// TIA Portal project "FactoryIO-ProductAllocate" (V17)

(* hardware
DEVICE "S71500/ET200MP-Station_1"  S7-1500 station
   slot 0: "Profilschiene_0"  6ES7 590-1***0-0AA0
   slot 1: "PLC_1"  CPU 1511-1 PN  6ES7 511-1AK00-0AB0  V1.8
   slot 2: "AI 8xU/I/RTD/TC ST_1"  AI 8xU/I/RTD/TC ST  6ES7 531-7KF00-0AB0  V2.0
   slot 3: "AI 8xU/I/RTD/TC ST_2"  AI 8xU/I/RTD/TC ST  6ES7 531-7KF00-0AB0  V2.0
   slot 4: "AI 8xU/I/RTD/TC ST_3"  AI 8xU/I/RTD/TC ST  6ES7 531-7KF00-0AB0  V2.0
   slot 5: "AI 8xU/I/RTD/TC ST_4"  AI 8xU/I/RTD/TC ST  6ES7 531-7KF00-0AB0  V2.0
   slot 6: "DI 16x24VDC BA_1"  DI 16x24VDC BA  6ES7 521-1BH10-0AA0  V1.0
DEVICE "PC station"  SIMATIC PC station
   slot 0: "PC station"  Rail  SIMATIC PC-Station  V1.0
      slot 125: "Stationmanager"  Station_Manager  V6.0.4
   slot 1: "IE general_1"  IE General  IE_CP  V8.2.0
      slot 1: "PROFINET interface"  IEGeneral.Interface.8.2.0
   slot 3: "HMI_RT_1"  WinCC RT Advanced  6AV2 104-0xxxx-xxxx  17.0.0.0
      slot 33792: "Computer interface"  Host interface
*)

// ===== PLC "PLC_1"  CPU 1511-1 PN =====

VAR_GLOBAL   // PLC tag table "Standard-Variablentabelle"
   "EMStop" AT %E0.0 : Bool;
   "Stop Button" AT %I0.1 : Bool;
   "Start Button" AT %I0.2 : Bool;
   "GreenSensor" AT %I0.3 : Bool;
   "BlueSensor" AT %I0.4 : Bool;
   "Konveyor1Motor" AT %Q0.0 : Bool;
   "Konveyor2Motor" AT %Q0.1 : Bool;
   "Konveyor3Motor" AT %Q0.2 : Bool;
   "Pusher1" AT %Q0.3 : Bool;
   "Pusher2" AT %Q0.4 : Bool;
   "StartLed" AT %Q0.5 : Bool;
   "StopLed" AT %Q0.6 : Bool;
   "GreenDisplay" AT %QW30 : Word;
   "BlueDisplay" AT %QW32 : Word;
   "MetalDisplay" AT %QW34 : Word;
   "Tag_1" AT %M20.1 : Bool;
   "Tag_2" AT %MD100 : DWord;
   "Tag_3" AT %MW30 : Int;
   "Tag_4" AT %M10.0 : Bool;
   "Tag_5" AT %M10.1 : Bool;
   "Tag_6" AT %MW32 : Int;
   "Tag_7" AT %MW34 : Int;
   "MetalSensor" AT %I0.5 : Bool;
   "Tag_8" AT %M10.2 : Bool;
   "Emitter" AT %Q0.7 : Bool;
   "Tag_9" AT %QD30 : DWord;
   "Tag_10" AT %QD32 : DWord;
   "Tag_11" AT %QD34 : DWord;
END_VAR

// folder: System blocks/Program resources

DATA_BLOCK "IEC_Counter_0_DB"   // DB1
{ S7_Optimized_Access := 'TRUE' }
AUTHOR : Simatic
FAMILY : IEC
NAME : CNTR
VERSION : 1.0
// stored: InstanceOfName IEC_COUNTER
"IEC_COUNTER"
BEGIN
END_DATA_BLOCK

DATA_BLOCK "IEC_Counter_0_DB_1"   // DB2
{ S7_Optimized_Access := 'TRUE' }
AUTHOR : Simatic
FAMILY : IEC
NAME : CNTR
VERSION : 1.0
// stored: InstanceOfName IEC_COUNTER
"IEC_COUNTER"
BEGIN
END_DATA_BLOCK

DATA_BLOCK "IEC_Counter_0_DB_2"   // DB3
{ S7_Optimized_Access := 'TRUE' }
AUTHOR : Simatic
FAMILY : IEC
NAME : CNTR
VERSION : 1.0
// stored: InstanceOfName IEC_COUNTER
"IEC_COUNTER"
BEGIN
END_DATA_BLOCK

// folder: (top level)

FUNCTION "MHJ-PLC-Lab-Function-S71500" : Void   // FC9000, SCL
{ S7_Optimized_Access := 'TRUE' }
VERSION : 0.1
   VAR_TEMP
      Value : Byte;
      ForCounter : Int;
   END_VAR
   VAR CONSTANT
      Value_01_DW : DWord := 16#1223_5486;
      Value_02_DW : DWord := 16#A6C9_D1F5;
   END_VAR
BEGIN

   #Value:=PEEK(area := 16#82,
        dbNumber := 0,
        byteOffset := 511);
   #Value := #Value + 1;

   POKE(area := 16#82,
        dbNumber := 0,
        byteOffset := 511,
        value := #Value);

   POKE(area := 16#82,
        dbNumber := 0,
        byteOffset := 1016,
        value := #Value_01_DW);
   POKE(area := 16#82,
        dbNumber := 0,
        byteOffset := 1020,
        value := #Value_02_DW);

   FOR #ForCounter := 0 TO 63 DO
       #Value:=PEEK(area := 16#1,
            dbNumber := 0,
            byteOffset := #ForCounter);
       POKE(area := 16#81,
            dbNumber := 0,
            byteOffset := #ForCounter,
            value := #Value);
   END_FOR;
   #Value := PEEK(area := 16#1,
                  dbNumber := 0,
                  byteOffset := 512);
   POKE(area := 16#82,
        dbNumber := 0,
        byteOffset := 512,
        value := #Value);
END_FUNCTION

ORGANIZATION_BLOCK "Main"   // OB1, LAD, ProgramCycle
TITLE = "Main Program Sweep (Cycle)"
{ S7_Optimized_Access := 'TRUE' }
VERSION : 0.1
   VAR_INPUT
      Initial_Call : Bool;   // Initial call of this OB
      Remanence : Bool;   // =True, if remanent data are available
   END_VAR
   VAR_TEMP   // added for the SCL form of the ladder/FBD networks
      _w1 : Bool;
   END_VAR
BEGIN

REGION Network 1
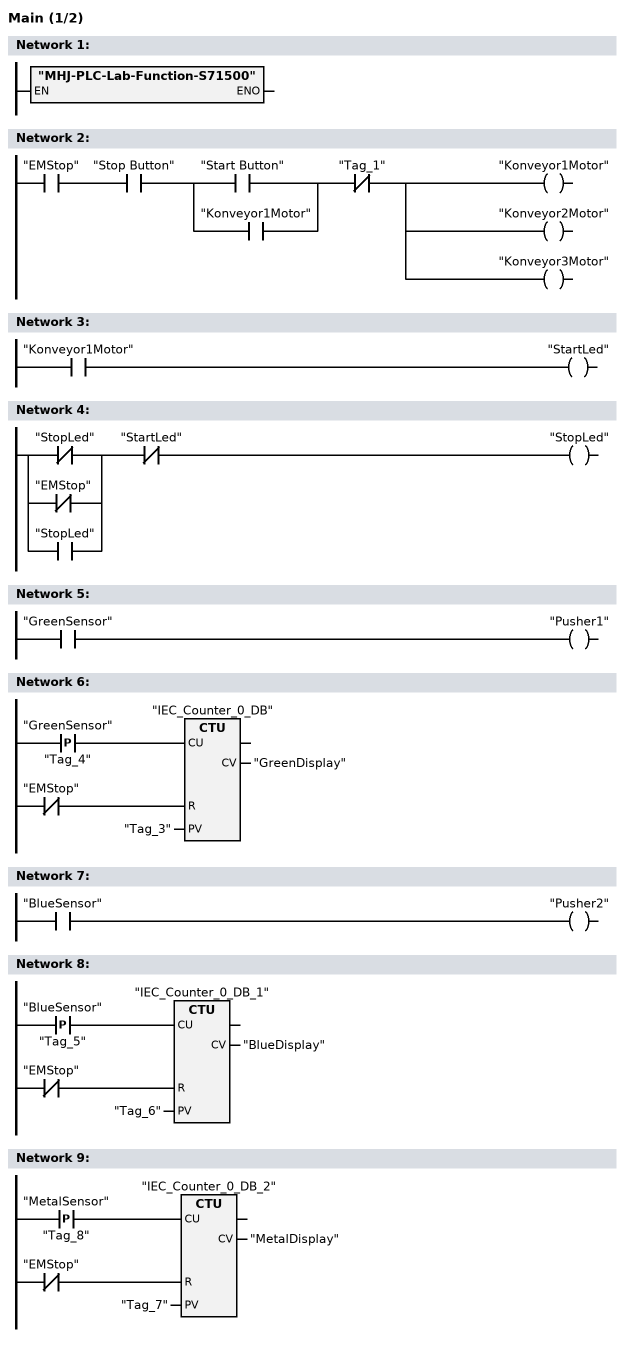
   RUNG wire#powerrail
      "MHJ-PLC-Lab-Function-S71500"()
   END_RUNG
   // the same network as SCL:
   "MHJ-PLC-Lab-Function-S71500"();
END_REGION

REGION Network 2
   RUNG wire#powerrail
      Contact( "EMStop" )
      Contact( "Stop Button" )
      wire#w1
      Contact( "Start Button" )
      wire#w2
      I_Contact( "Tag_1" )
      wire#w3
      Coil( "Konveyor1Motor" )
   END_RUNG
   RUNG wire#w1
      Contact( "Konveyor1Motor" )
   END_RUNG wire#w2
   RUNG wire#w3
      Coil( "Konveyor2Motor" )
   END_RUNG
   RUNG wire#w3
      Coil( "Konveyor3Motor" )
   END_RUNG
   // the same network as SCL:
   "Konveyor1Motor" := "EMStop" AND "Stop Button" AND ("Start Button" OR "Konveyor1Motor") AND NOT "Tag_1";
   "Konveyor2Motor" := "Konveyor1Motor";
   "Konveyor3Motor" := "Konveyor1Motor";
END_REGION

REGION Network 3
   RUNG wire#powerrail
      Contact( "Konveyor1Motor" )
      Coil( "StartLed" )
   END_RUNG
   // the same network as SCL:
   "StartLed" := "Konveyor1Motor";
END_REGION

REGION Network 4
   RUNG wire#powerrail
      I_Contact( "StopLed" )
      wire#w1
      I_Contact( "StartLed" )
      Coil( "StopLed" )
   END_RUNG
   RUNG wire#powerrail
      I_Contact( "EMStop" )
   END_RUNG wire#w1
   RUNG wire#powerrail
      Contact( "StopLed" )
   END_RUNG wire#w1
   // the same network as SCL:
   "StopLed" := (NOT "StopLed" OR NOT "EMStop" OR "StopLed") AND NOT "StartLed";
END_REGION

REGION Network 5
   RUNG wire#powerrail
      Contact( "GreenSensor" )
      Coil( "Pusher1" )
   END_RUNG
   // the same network as SCL:
   "Pusher1" := "GreenSensor";
END_REGION

REGION Network 6
   #_w1 := "GreenSensor" AND NOT "Tag_4";   // rising edge of "GreenSensor"
   "Tag_4" := "GreenSensor";
   "IEC_Counter_0_DB".CTU(CU := #_w1, R := NOT "EMStop", PV := "Tag_3", CV => "GreenDisplay");
END_REGION

REGION Network 7
   RUNG wire#powerrail
      Contact( "BlueSensor" )
      Coil( "Pusher2" )
   END_RUNG
   // the same network as SCL:
   "Pusher2" := "BlueSensor";
END_REGION

REGION Network 8
   #_w1 := "BlueSensor" AND NOT "Tag_5";   // rising edge of "BlueSensor"
   "Tag_5" := "BlueSensor";
   "IEC_Counter_0_DB_1".CTU(CU := #_w1, R := NOT "EMStop", PV := "Tag_6", CV => "BlueDisplay");
END_REGION

REGION Network 9
   #_w1 := "MetalSensor" AND NOT "Tag_8";   // rising edge of "MetalSensor"
   "Tag_8" := "MetalSensor";
   "IEC_Counter_0_DB_2".CTU(CU := #_w1, R := NOT "EMStop", PV := "Tag_7", CV => "MetalDisplay");
END_REGION

REGION Network 10
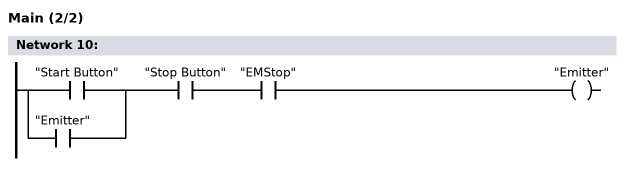
   RUNG wire#powerrail
      Contact( "Start Button" )
      wire#w1
      Contact( "Stop Button" )
      Contact( "EMStop" )
      Coil( "Emitter" )
   END_RUNG
   RUNG wire#powerrail
      Contact( "Emitter" )
   END_RUNG wire#w1
   // the same network as SCL:
   "Emitter" := ("Start Button" OR "Emitter") AND "Stop Button" AND "EMStop";
END_REGION
END_ORGANIZATION_BLOCK

(* ===== HMI "HMI_RT_1" =====
system functions are stored by id; their names below are inferred from use
connection "HMI_Connection_1": ETHERNET, S7_1500_OMS

HMI tags "Default tag table"
   "GreenDisplay" : Word = PLC GreenDisplay AT %QW30, 1 s
   "Pusher1" : Bool = PLC Pusher1 AT %Q0.3, 1 s
   "BlueDisplay" : Word = PLC BlueDisplay AT %QW32, 1 s
   "MetalDisplay" : Word = PLC MetalDisplay AT %QW34, 1 s
   "Konveyor1Motor" : Bool = PLC Konveyor1Motor AT %Q0.0, 1 s
   "Start Button" : Bool = PLC "Start Button" AT %I0.2, 1 s
   "Stop Button" : Bool = PLC "Stop Button" AT %I0.1, 1 s
   "EMStop" : Bool = PLC EMStop AT %I0.0, 1 s
   "StopLed" : Bool = PLC StopLed AT %Q0.6, 1 s
   "StartLed" : Bool = PLC StartLed AT %Q0.5, 1 s
   "Pusher2" : Bool = PLC Pusher2 AT %Q0.4, 1 s
   "MetalSensor" : Bool = PLC MetalSensor AT %I0.5, 1 s

screen "Screen_1" 600x800
   Button "Button_1" at 126,21 size 96x32; TextOff 'START'
      on Click: SetBit("Start Button")
   Button "Button_2" at 369,21 size 96x32; TextOff 'STOP'
      on Click: SetBit("Stop Button")
   Button "Button_3" at 249,21 size 96x32; TextOff 'EMSTOP'
      on Click: SetBit("EMStop")
   IOField "I/O field_1" at 361,175 size 70x43; FormatPattern 99
      ProcessValue <- "GreenDisplay"
   SymbolLibrary "Symbol library_1" at 57,176 size 271x42
      Appearance <- "Pusher1"
   TextField "Text field_1" at 150,123 size 287x29; Text 'GREEN PUSHER & DISPLAY'
   IOField "I/O field_2" at 361,294 size 70x43; FormatPattern 99
      ProcessValue <- "BlueDisplay"
   SymbolLibrary "Symbol library_2" at 57,295 size 271x42
      Appearance <- "Pusher2"
   TextField "Text field_2" at 150,242 size 287x29; Text 'BLUE PUSHER & DISPLAY'
   IOField "I/O field_3" at 361,413 size 70x43; FormatPattern 99
      ProcessValue <- "MetalDisplay"
   SymbolLibrary "Symbol library_3" at 57,414 size 271x42
   TextField "Text field_3" at 150,361 size 287x29; Text 'METAL PUSHER & DISPLAY'
   SymbolLibrary "Symbol library_4" at 56,536 size 433x166
      Appearance <- "Konveyor1Motor"
   TextField "Text field_4" at 150,483 size 224x39; Text 'KONVEYOR ON/OFF'
   Circle "Circle_1" at 489,295 size 48x48
      Appearance <- "Pusher2"
   Circle "Circle_2" at 489,170 size 48x48
      Appearance <- "Pusher1"
   Circle "Circle_3" at 489,408 size 48x48
      Appearance <- "MetalSensor"
   Circle "Circle_4" at 150,63 size 48x48
      Appearance <- "StartLed"
   Circle "Circle_5" at 389,63 size 48x48
      Appearance <- "StopLed"
*)